(* Logix 5000 project; controller Transcat vendor 1 type 14 code 152 rev 32.11; software revision 32.02; part 3 of 3 *)
(* tags used below, declared in another part *)
   AllDeviceEnable : BOOL;   // A bit to enable or disable the running of all devices
   alwaysOFF : BOOL;
   AlwaysOFF2 : BOOL;
   Device : Device[20];
   RecipeStart : BOOL;   // Bit to start and stop a recipe execution
   VF201 : Acrison_Feeder;   // Small Feeder 2 Tags
(* MainProgram, continued *)

ROUTINE VF201_Small_Feeder_2_AcrisonVFD   (* ladder *)
// Small Feeder 2 - Control via PowerFlex 525 VFD
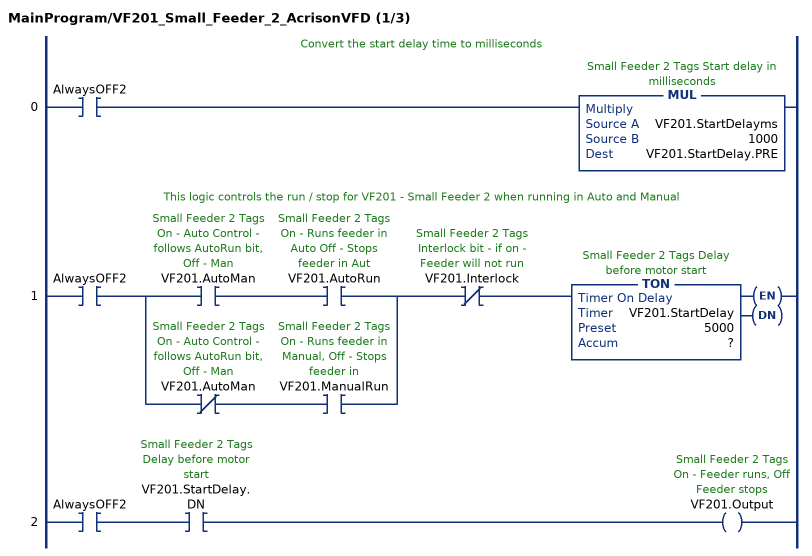
   // Convert the start delay time to milliseconds
   0: XIC(AlwaysOFF2)MUL(VF201.StartDelayms,1000,VF201.StartDelay.PRE);
   // This logic controls the run / stop for VF201 - Small Feeder 2 when running in Auto and Manual
   1: XIC(AlwaysOFF2)[XIC(VF201.AutoMan) XIC(VF201.AutoRun) ,XIO(VF201.AutoMan) XIC(VF201.ManualRun) ]XIO(VF201.Interlock)TON(VF201.StartDelay,?,?);
   2: XIC(AlwaysOFF2)XIC(VF201.StartDelay.DN)OTE(VF201.Output);
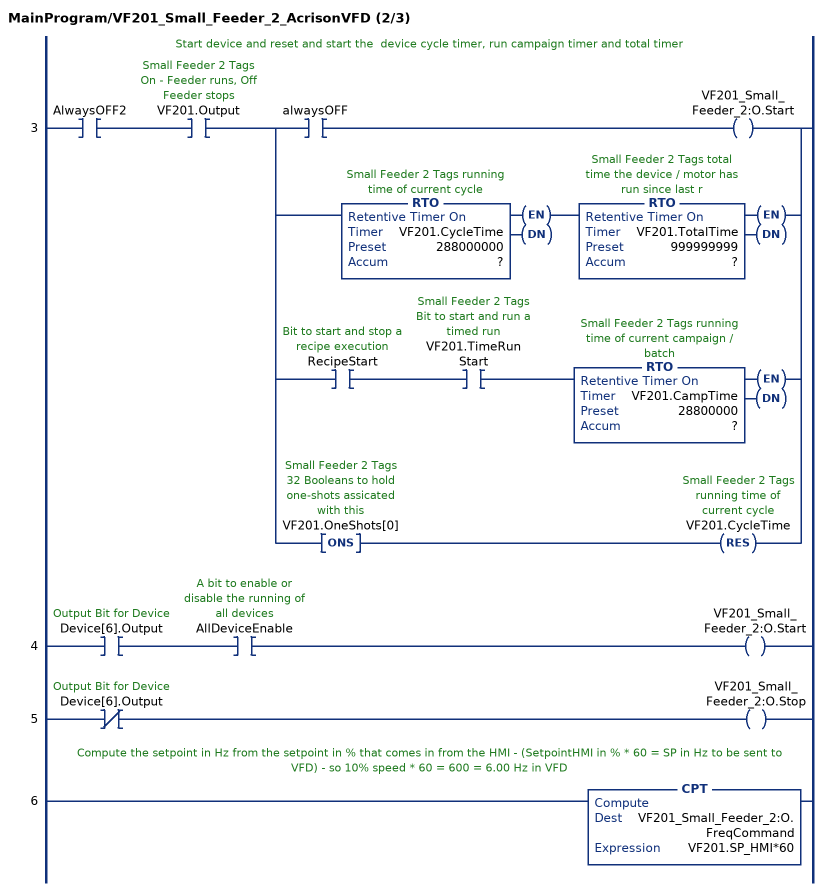
   // Start device and reset and start the  device cycle timer, run campaign timer and total timer
   3: XIC(AlwaysOFF2)XIC(VF201.Output)[XIC(alwaysOFF) OTE(VF201_Small_Feeder_2:O.Start) ,[RTO(VF201.CycleTime,?,?) RTO(VF201.TotalTime,?,?) ,XIC(RecipeStart) XIC(VF201.TimeRunStart) RTO(VF201.CampTime,?,?) ,ONS(VF201.OneShots[0]) RES(VF201.CycleTime) ] ];
   4: XIC(Device[6].Output)XIC(AllDeviceEnable)OTE(VF201_Small_Feeder_2:O.Start);
   5: XIO(Device[6].Output)OTE(VF201_Small_Feeder_2:O.Stop);
   // Compute the setpoint in Hz from the setpoint in % that comes in from the HMI - (SetpointHMI in % * 60 = SP in Hz to be sent to VFD) - so 10% speed * 60 = 600 = 6.00 Hz in VFD
   6: CPT(VF201_Small_Feeder_2:O.FreqCommand,VF201.SP_HMI*60);
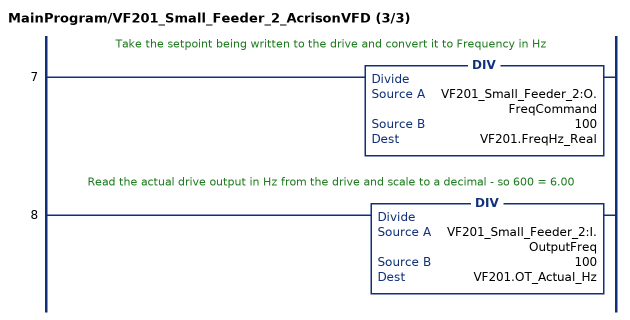
   // Take the setpoint being written to the drive and convert it to Frequency in Hz
   7: DIV(VF201_Small_Feeder_2:O.FreqCommand,100,VF201.FreqHz_Real);
   // Read the actual drive output in Hz from the drive and scale to a decimal - so 600 = 6.00
   8: DIV(VF201_Small_Feeder_2:I.OutputFreq,100,VF201.OT_Actual_Hz);
END_ROUTINE
END_PROGRAM
